PROGRAM prgCom
VAR
	fbCom			: FB_MqttCommunicator;
	byte_array : ARRAY[0..1023] OF BYTE;
	struct_transfer	: struct_ADS_Auhofcenter;
	mSize_to_Big: BOOL;
	uint_size: UINT;
END_VAR

fbCom(
	bConnect:= TRUE, 
	sUserName:= '820ed295-9a22-4ba6-b6eb-7ebc44129c59', 
	sUserPassword:= '61ffcacb-a97f-4d5a-a14e-16ed8c97a18f', 
	eSavePositionCertificate:= eSavePositionOnPLC.ePostionC, 
	bConnected=> , 
	bError=> , 
	hrErrorCode=> , 
	eConnectionState=> , 
	eErrorMessage_Out=> );
	
// copy values to struct	
struct_transfer.int_liveCount 				:= struct_transfer.int_liveCount+1;
struct_transfer.rHeartbeat			:= MAIN.rHeartbeat ;
struct_transfer.rErrorWarning		:= MAIN.rErrorWarning ;
struct_transfer.rSPOptReady			:= MAIN.rSPOptReady ;
struct_transfer.rUmfVorlaufSek		:= MAIN.rUmfVorlaufSek ;
struct_transfer.rUmfRuecklaufSek	:=  MAIN.rUmfRuecklaufSek;
struct_transfer.bPumpenState		:= MAIN.bPumpenState ;
struct_transfer.rRTMall_EG_Billa	:= MAIN.rRTMall_EG_Billa ;
struct_transfer.rRTMall_EG_RichutngBT2	:= MAIN.rRTMall_EG_RichutngBT2 ;
struct_transfer.rRTMall_EG_VorPost	:=  MAIN.rRTMall_EG_VorPost;
struct_transfer.rRTMall_OG_Nordseitig :=  MAIN.rRTMall_OG_Nordseitig;
struct_transfer.rRTMall_OG_Suedseitig := MAIN.rRTMall_OG_Suedseitig ;
struct_transfer.rRTMall_OG_VorTKMaxx := MAIN.rRTMall_OG_VorTKMaxx ;
struct_transfer.rRTMall_OG_VorStrasslSchaider :=  MAIN.rRTMall_OG_VorStrasslSchaider;
struct_transfer.rNewTargetValue		:= MAIN.rNewTargetValue ;
struct_transfer.rBT2UmfVorlaufSek	:= MAIN.rBT2UmfVorlaufSek ;
struct_transfer.rBT2UmfRuecklaufPri	:= MAIN.rBT2UmfRuecklaufPri ;
struct_transfer.bBT2PumpenState		:=  MAIN.bBT2PumpenState;
struct_transfer.rBT2RTMall_EG_Nord	:= MAIN.rBT2RTMall_EG_Nord ;
struct_transfer.rBT2RTMall_OG_Nord	:= MAIN.rBT2RTMall_OG_Nord ;
struct_transfer.rBT2RTMall_EG_Sued	:= MAIN.rBT2RTMall_EG_Sued ;
struct_transfer.rBT2RTMall_OG_Sued	:= MAIN.rBT2RTMall_OG_Sued ;
struct_transfer.rBT2NewTargetValue	:= MAIN.rBT2NewTargetValue ;
struct_transfer.rBT3UmfVorlaufSek	:= MAIN.rBT3UmfVorlaufSek ;
struct_transfer.rBT3UmfRuecklaufSek	:= MAIN.rBT3UmfRuecklaufSek ;
struct_transfer.bBT3PumpenState		:= MAIN.bBT3PumpenState ;
struct_transfer.rBT3RTMall_EG_West	:= MAIN.rBT3RTMall_EG_West ;
struct_transfer.rBT3RTMall_OG_West	:= MAIN.rBT3RTMall_OG_West ;
struct_transfer.rBT3RTMall_EG_HK31	:= MAIN.rBT3RTMall_EG_HK31 ;
struct_transfer.rBT3RTMall_EG_HK32	:= MAIN.rBT3RTMall_EG_HK32 ;
struct_transfer.rBT3RTMall_OG_K33	:= MAIN.rBT3RTMall_OG_K33 ;
struct_transfer.rBT3RTMall_OG_K34	:= MAIN.rBT3RTMall_OG_K34 ;
struct_transfer.rBT3RTMall_OG_Ost	:= MAIN.rBT3RTMall_OG_Ost ;
struct_transfer.rBT3RTMall_EG_Ost	:=  MAIN.rBT3RTMall_EG_Ost;
struct_transfer.rBT3RTMall_EG_HK35	:= MAIN.rBT3RTMall_EG_HK35 ;
struct_transfer.rBT3RTMall_OG_HK37	:= MAIN.rBT3RTMall_OG_HK37 ;
struct_transfer.rBT3NewTargetValue	:= MAIN.rBT3NewTargetValue ;
struct_transfer.rBT4UmfVorlaufSek	:= MAIN.rBT4UmfVorlaufSek ;
struct_transfer.rBT4UmfRuecklaufSek	:= MAIN.rBT4UmfRuecklaufSek ;
struct_transfer.bBT4PumpenState		:= MAIN.bBT4PumpenState ;
struct_transfer.rBT4RTMall_EG		:= MAIN.rBT4RTMall_EG ;
struct_transfer.rBT5RTMall_OG		:= MAIN.rBT5RTMall_OG ;
struct_transfer.rBT6RTMall_OG		:= MAIN.rBT6RTMall_OG ;
struct_transfer.rBT6RTMall_EG		:= MAIN.rBT6RTMall_EG ;
struct_transfer.rBT4NewTargetValue	:= MAIN.rBT4NewTargetValue ;
struct_transfer.rAussentemperatur	:= MAIN.rAussentemperatur ;
struct_transfer.bEnableOp			:= MAIN.bEnableOp ;
struct_transfer.bSEnableOp			:= MAIN.bSEnableOp ;
struct_transfer.bEnableOpBT2		:= MAIN.bEnableOpBT2 ;
struct_transfer.bSEnableOpBT2		:= MAIN.bSEnableOpBT2 ;
struct_transfer.bEnableOpBT3		:= MAIN.bEnableOpBT3 ;
struct_transfer.bSEnableOpBT3		:= MAIN.bSEnableOpBT3 ;
struct_transfer.bEnableOpBT4		:= MAIN.bEnableOpBT4 ;
struct_transfer.bSEnableOpBT4		:= MAIN.bSEnableOpBT4 ;
struct_transfer.rBT1EM_Power_kW		:= MAIN.rBT1EM_Power_kW ;
struct_transfer.lrBT1EM_Counter_kWh	:= MAIN.lrBT1EM_Counter_kWh ;
struct_transfer.rBT2EM_Power_kW		:= MAIN.rBT2EM_Power_kW ;
struct_transfer.lrBT2EM_Counter_kWh	:= MAIN.lrBT2EM_Counter_kWh ;
struct_transfer.rBT3EM_Power_kW		:= MAIN.rBT3EM_Power_kW ;
struct_transfer.lrBT3EM_Counter_kWh	:= MAIN.lrBT3EM_Counter_kWh ;
struct_transfer.rBT4EM_Power_kW		:= MAIN.rBT4EM_Power_kW ;
struct_transfer.lrBT4EM_Counter_kWh	:= MAIN.lrBT4EM_Counter_kWh ;
struct_transfer.lrPowerPV_1_1		:= prgPV.lrPowerPV_1_1 ;
struct_transfer.lrPowerPV_1_2		:= prgPV.lrPowerPV_1_2 ;
struct_transfer.lrPowerPV_2_1		:= prgPV.lrPowerPV_2_1 ;
struct_transfer.lrPowerPV_2_2		:= prgPV.lrPowerPV_2_2 ;
struct_transfer.lrPowerPV_3_1		:= prgPV.lrPowerPV_3_1 ;
struct_transfer.lrPowerPV_3_2		:= prgPV.lrPowerPV_3_2 ;
struct_transfer.lrPowerPV_3_3		:= prgPV.lrPowerPV_3_3 ;
struct_transfer.lrPowerPV_3_4		:= prgPV.lrPowerPV_3_4 ;
struct_transfer.lrPowerPV_3_5		:= prgPV.lrPowerPV_3_5 ;
struct_transfer.lrPowerPV_3_6		:= prgPV.lrPowerPV_3_6 ;
struct_transfer.lrPowerPV			:= prgPV.lrPowerPV ;
struct_transfer.rUmfVorlaufPri		:=  MAIN.rUmfVorlaufPri;
struct_transfer.rUmfRuecklaufPri	:=  Main.rUmfRuecklaufPri;
struct_transfer.rBT3UmfRuecklaufPri		:= MAIN.rBT3UmfRuecklaufPri ;
struct_transfer.rBT3UmfVorlaufPri		:= MAIN.rBT3UmfVorlaufPri ;
struct_transfer.rBT4UmfVorlaufPri		:=  Main.rBT4UmfVorlaufPri;
struct_transfer.rBT4UmfRuecklaufPri		:= MAIN.rBT4UmfRuecklaufPri ;
(*struct_transfer.		:=  ;
struct_transfer.		:=  ;
struct_transfer.		:=  ;
struct_transfer.		:=  ;
struct_transfer.		:=  ;
struct_transfer.		:=  ;
*)

// copy struct to byte array
IF SIZEOF(struct_transfer) > SIZEOF(byte_array) THEN
	memcpy(ADR(byte_array),ADR(struct_transfer),SIZEOF(byte_array));
	uint_size := SIZEOF(struct_transfer);
	mSize_to_Big := TRUE;
ELSE
	memcpy(ADR(byte_array),ADR(struct_transfer),SIZEOF(struct_transfer));
	mSize_to_Big := FALSE;
END_IF
uint_size := SIZEOF(struct_transfer);

END_PROGRAM

(* stored: Version 1.1.0.1, ProductVersion 3.1.4024.12
   POU prgCom: Id {27ef1611-e16c-4e06-8ec4-cfa9c8ffb71b}, SpecialFunc None *)
